// TIA Portal V17 export
// export: Created 2021-12-03T08:08:05.7344229Z, ExportSetting WithDefaults, DisplayName Totally Integrated Automation Portal, DisplayVersion V17, DisplayName TIA Portal Openness, DisplayVersion V17, DisplayName TIA Portal Version Control Interface, DisplayVersion V17, DisplayName STEP 7 Professional, DisplayVersion V17, DisplayName STEP 7 Safety, DisplayVersion V17, DisplayName WinCC Advanced, DisplayVersion V17
VAR_GLOBAL   // PLC tag table "Data_Send"
   CircBrcSts AT %MW100 : Int;   // Автоматические выключатели
   CircBrcSts_0 AT %M100.0 : Bool;
   CircBrcSts_1 AT %M100.1 : Bool;
   CircBrcSts_2 AT %M100.2 : Bool;
   CircBrcSts_3 AT %M100.3 : Bool;
   CircBrcSts_4 AT %M100.4 : Bool;
   CircBrcSts_5 AT %M100.5 : Bool;
   CircBrcSts_6 AT %M100.6 : Bool;
   CircBrcSts_7 AT %M100.7 : Bool;
   CircBrcSts_8 AT %M101.0 : Bool;
   CircBrcSts_9 AT %M101.1 : Bool;
   CircBrcSts_10 AT %M101.2 : Bool;
   CircBrcSts_11 AT %M101.3 : Bool;
   CircBrcSts_12 AT %M101.4 : Bool;
   CircBrcSts_13 AT %M101.5 : Bool;
   CircBrcSts_14 AT %M101.6 : Bool;
   CircBrcSts_15 AT %M101.7 : Bool;
   AccSts AT %MW102 : Int;   // Сигналы с ускорителя
   AccSts_0 AT %M102.0 : Bool;
   AccSts_1 AT %M102.1 : Bool;
   AccSts_2 AT %M102.2 : Bool;
   AccSts_3 AT %M102.3 : Bool;
   AccSts_4 AT %M102.4 : Bool;
   AccSts_5 AT %M102.5 : Bool;
   AccSts_6 AT %M102.6 : Bool;
   AccSts_7 AT %M102.7 : Bool;
   AccSts_8 AT %M103.0 : Bool;
   AccSts_9 AT %M103.1 : Bool;
   AccSts_10 AT %M103.2 : Bool;
   AccSts_11 AT %M103.3 : Bool;
   AccSts_12 AT %M103.4 : Bool;
   AccSts_13 AT %M103.5 : Bool;
   AccSts_14 AT %M103.6 : Bool;
   AccSts_15 AT %M103.7 : Bool;
   P1EmrStp AT %MW104 : Int;   // Аварийный останов Р1
   P1EmrStp_0 AT %M104.0 : Bool;
   P1EmrStp_1 AT %M104.1 : Bool;
   P1EmrStp_2 AT %M104.2 : Bool;
   P2EmrStp AT %MW106 : Int;   // Аварийный останов Р2
   P2EmrStp_0 AT %M106.0 : Bool;
   P2EmrStp_1 AT %M106.1 : Bool;
   P2EmrStp_2 AT %M106.2 : Bool;
   P3EmrStp AT %MW108 : Int;   // Аварийный останов Р3
   P3EmrStp_0 AT %M108.0 : Bool;
   P3EmrStp_1 AT %M108.1 : Bool;
   P3EmrStp_2 AT %M108.2 : Bool;
   AccEmrStp AT %MW110 : Int;   // Аварийный останов от ускорителя
   AccEmrStp_0 AT %M110.0 : Bool;
   AccEmrStp_1 AT %M110.1 : Bool;
   AccEmrStp_2 AT %M110.2 : Bool;
   DosimEmrStp AT %MW112 : Int;   // Аварийный останов от дозиметра
   DosimEmrStp_0 AT %M112.0 : Bool;
   DosimEmrStp_1 AT %M112.1 : Bool;
   DosimEmrStp_2 AT %M112.2 : Bool;
   Cmd AT %MW114 : Int;   // Состояние системы
   Cmd_0 AT %M114.0 : Bool;
   Cmd_1 AT %M114.1 : Bool;
   Cmd_2 AT %M114.2 : Bool;
   Cmd_3 AT %M114.3 : Bool;
   Cmd_4 AT %M114.4 : Bool;
   Cmd_5 AT %M114.5 : Bool;
   Cmd_6 AT %M114.6 : Bool;
   Cmd_7 AT %M114.7 : Bool;
   Cmd_8 AT %M115.0 : Bool;
   Cmd_9 AT %M115.1 : Bool;
   Cmd_10 AT %M115.2 : Bool;
   Cmd_11 AT %M115.3 : Bool;
   Cmd_12 AT %M115.4 : Bool;
   Cmd_13 AT %M115.5 : Bool;
   Cmd_14 AT %M115.6 : Bool;
   Cmd_15 AT %M115.7 : Bool;
   Sft AT %MW116 : Int;   // Состояние систем безопасности
   Sft_0 AT %M116.0 : Bool;
   Sft_1 AT %M116.1 : Bool;
   Sft_2 AT %M116.2 : Bool;
   Sft_3 AT %M116.3 : Bool;
   Sft_4 AT %M116.4 : Bool;
   Sft_5 AT %M116.5 : Bool;
   Sft_6 AT %M116.6 : Bool;
   Sft_7 AT %M116.7 : Bool;
   Sft_8 AT %M117.0 : Bool;
   Sft_9 AT %M117.1 : Bool;
   Sft_10 AT %M117.2 : Bool;
   Sft_11 AT %M117.3 : Bool;
   Sft_12 AT %M117.4 : Bool;
   Sft_13 AT %M117.5 : Bool;
   Sft_14 AT %M117.6 : Bool;
   Sft_15 AT %M117.7 : Bool;
   GnEmStp AT %MW118 : Int;
   GnEmStp_0 AT %M118.0 : Bool;
   GnEmStp_1 AT %M118.1 : Bool;
   GnEmStp_2 AT %M118.2 : Bool;
   Mod400_RlyOn AT %MW120 : Int;
   Mod400_RlyOn_0 AT %M120.0 : Bool;
   Mod400_RlyOn_1 AT %M120.1 : Bool;
   Mod400_RlyOn_2 AT %M120.2 : Bool;
   Mod400_RlyOn_3 AT %M120.3 : Bool;
   Mod400_RlyOn_4 AT %M120.4 : Bool;
   Mod400_RlyOn_5 AT %M120.5 : Bool;
   Mod400_RlyOn_6 AT %M120.6 : Bool;
   Mod400_RlyOn_7 AT %M120.7 : Bool;
   Mod400_RlyOn_8 AT %M121.0 : Bool;
   Mod400_RlyOn_9 AT %M121.1 : Bool;
   Mod400_RlyOn_10 AT %M121.2 : Bool;
   Mod400_RlyOn_11 AT %M121.3 : Bool;
   Mod400_RlyOn_12 AT %M121.4 : Bool;
   Mod400_RlyOn_13 AT %M121.5 : Bool;
   Mod400_RlyOn_14 AT %M121.6 : Bool;
   Mod400_RlyOn_15 AT %M121.7 : Bool;
   Mod230_RlyOn AT %MW122 : Int;
   Mod230_RlyOn_0 AT %M122.0 : Bool;
   Mod230_RlyOn_1 AT %M122.1 : Bool;
   Mod230_RlyOn_2 AT %M122.2 : Bool;
   Mod230_RlyOn_3 AT %M122.3 : Bool;
   Mod230_RlyOn_4 AT %M122.4 : Bool;
   Mod230_RlyOn_5 AT %M122.5 : Bool;
   Mod230_RlyOn_6 AT %M122.6 : Bool;
   Mod230_RlyOn_7 AT %M122.7 : Bool;
   Mod230_RlyOn_8 AT %M123.0 : Bool;
   Mod230_RlyOn_9 AT %M123.1 : Bool;
   Mod230_RlyOn_10 AT %M123.2 : Bool;
   Mod230_RlyOn_11 AT %M123.3 : Bool;
   Mod230_RlyOn_12 AT %M123.4 : Bool;
   Mod230_RlyOn_13 AT %M123.5 : Bool;
   Mod230_RlyOn_14 AT %M123.6 : Bool;
   Mod230_RlyOn_15 AT %M123.7 : Bool;
   Chill_RlyOn AT %MW124 : Int;
   Chill_RlyOn_0 AT %M124.0 : Bool;
   Chill_RlyOn_1 AT %M124.1 : Bool;
   Chill_RlyOn_2 AT %M124.2 : Bool;
   Chill_RlyOn_3 AT %M124.3 : Bool;
   Chill_RlyOn_4 AT %M124.4 : Bool;
   Chill_RlyOn_5 AT %M124.5 : Bool;
   Chill_RlyOn_6 AT %M124.6 : Bool;
   Chill_RlyOn_7 AT %M124.7 : Bool;
   Chill_RlyOn_8 AT %M125.0 : Bool;
   Chill_RlyOn_9 AT %M125.1 : Bool;
   Chill_RlyOn_10 AT %M125.2 : Bool;
   Chill_RlyOn_11 AT %M125.3 : Bool;
   Chill_RlyOn_12 AT %M125.4 : Bool;
   Chill_RlyOn_13 AT %M125.5 : Bool;
   Chill_RlyOn_14 AT %M125.6 : Bool;
   Chill_RlyOn_15 AT %M125.7 : Bool;
   Acc_RlyOn AT %MW126 : Int;
   Acc_RlyOn_0 AT %M126.0 : Bool;
   Acc_RlyOn_1 AT %M126.1 : Bool;
   Acc_RlyOn_2 AT %M126.2 : Bool;
   Acc_RlyOn_3 AT %M126.3 : Bool;
   Acc_RlyOn_4 AT %M126.4 : Bool;
   Acc_RlyOn_5 AT %M126.5 : Bool;
   Acc_RlyOn_6 AT %M126.6 : Bool;
   Acc_RlyOn_7 AT %M126.7 : Bool;
   Acc_RlyOn_8 AT %M127.0 : Bool;
   Acc_RlyOn_9 AT %M127.1 : Bool;
   Acc_RlyOn_10 AT %M127.2 : Bool;
   Acc_RlyOn_11 AT %M127.3 : Bool;
   Acc_RlyOn_12 AT %M127.4 : Bool;
   Acc_RlyOn_13 AT %M127.5 : Bool;
   Acc_RlyOn_14 AT %M127.6 : Bool;
   Acc_RlyOn_15 AT %M127.7 : Bool;
   Conv_RlyOn AT %MW128 : Int;
   Conv_RlyOn_0 AT %M128.0 : Bool;
   Conv_RlyOn_1 AT %M128.1 : Bool;
   Conv_RlyOn_2 AT %M128.2 : Bool;
   Conv_RlyOn_3 AT %M128.3 : Bool;
   Conv_RlyOn_4 AT %M128.4 : Bool;
   Conv_RlyOn_5 AT %M128.5 : Bool;
   Conv_RlyOn_6 AT %M128.6 : Bool;
   Conv_RlyOn_7 AT %M128.7 : Bool;
   Conv_RlyOn_8 AT %M129.0 : Bool;
   Conv_RlyOn_9 AT %M129.1 : Bool;
   Conv_RlyOn_10 AT %M129.2 : Bool;
   Conv_RlyOn_11 AT %M129.3 : Bool;
   Conv_RlyOn_12 AT %M129.4 : Bool;
   Conv_RlyOn_13 AT %M129.5 : Bool;
   Conv_RlyOn_14 AT %M129.6 : Bool;
   Conv_RlyOn_15 AT %M129.7 : Bool;
   ConvSns AT %MW132 : Int;
   ConvSns_0 AT %M132.0 : Bool;
   ConvSns_1 AT %M132.1 : Bool;
   ConvSns_2 AT %M132.2 : Bool;
   ConvSns_3 AT %M132.3 : Bool;
   ConvSns_4 AT %M132.4 : Bool;
   ConvSns_5 AT %M132.5 : Bool;
   ConvSns_6 AT %M132.6 : Bool;
   ConvSns_7 AT %M132.7 : Bool;
   ConvSns_8 AT %M133.0 : Bool;
   ConvSns_9 AT %M133.1 : Bool;
   ConvSns_10 AT %M133.2 : Bool;
   ConvSns_11 AT %M133.3 : Bool;
   ConvSns_12 AT %M133.4 : Bool;
   ConvSns_13 AT %M133.5 : Bool;
   ConvSns_14 AT %M133.6 : Bool;
   ConvSns_15 AT %M133.7 : Bool;
   ScanSeq_Sts AT %MW134 : Int;
   ScanSeq_Sts_0 AT %M134.0 : Bool;
   ScanSeq_Sts_1 AT %M134.1 : Bool;
   ScanSeq_Sts_2 AT %M134.2 : Bool;
   ScanSeq_Sts_3 AT %M134.3 : Bool;
   ScanSeq_Sts_4 AT %M134.4 : Bool;
   ScanSeq_Sts_5 AT %M134.5 : Bool;
   ScanSeq_Sts_6 AT %M134.6 : Bool;
   ScanSeq_Sts_7 AT %M134.7 : Bool;
   ScanSeq_Sts_8 AT %M135.0 : Bool;
   ScanSeq_Sts_9 AT %M135.1 : Bool;
   ScanSeq_Sts_10 AT %M135.2 : Bool;
   ScanSeq_Sts_11 AT %M135.3 : Bool;
   ScanSeq_Sts_12 AT %M135.4 : Bool;
   ScanSeq_Sts_13 AT %M135.5 : Bool;
   ScanSeq_Sts_14 AT %M135.6 : Bool;
   ScanSeq_Sts_15 AT %M135.7 : Bool;
   DetLine_Sts AT %MW136 : Int;
   DetLine_Sts_0 AT %M136.0 : Bool;
   DetLine_Sts_1 AT %M136.1 : Bool;
   DetLine_Sts_2 AT %M136.2 : Bool;
   DetLine_Sts_3 AT %M136.3 : Bool;
   DetLine_Sts_4 AT %M136.4 : Bool;
   DetLine_Sts_5 AT %M136.5 : Bool;
   DetLine_Sts_6 AT %M136.6 : Bool;
   DetLine_Sts_7 AT %M136.7 : Bool;
   DetLine_Sts_8 AT %M137.0 : Bool;
   DetLine_Sts_9 AT %M137.1 : Bool;
   DetLine_Sts_10 AT %M137.2 : Bool;
   DetLine_Sts_11 AT %M137.3 : Bool;
   DetLine_Sts_12 AT %M137.4 : Bool;
   DetLine_Sts_13 AT %M137.5 : Bool;
   DetLine_Sts_14 AT %M137.6 : Bool;
   DetLine_Sts_15 AT %M137.7 : Bool;
   Pwr_All AT %MW138 : Int;
   Pwr_All_0 AT %M138.0 : Bool;
   Pwr_All_1 AT %M138.1 : Bool;
   Pwr_All_2 AT %M138.2 : Bool;
   Pwr_All_3 AT %M138.3 : Bool;
   Pwr_All_4 AT %M138.4 : Bool;
   Pwr_All_5 AT %M138.5 : Bool;
   Pwr_All_6 AT %M138.6 : Bool;
   Pwr_All_7 AT %M138.7 : Bool;
   Pwr_All_8 AT %M139.0 : Bool;
   Pwr_All_9 AT %M139.1 : Bool;
   Pwr_All_10 AT %M139.2 : Bool;
   Pwr_All_11 AT %M139.3 : Bool;
   Pwr_All_12 AT %M139.4 : Bool;
   Pwr_All_13 AT %M139.5 : Bool;
   Pwr_All_14 AT %M139.6 : Bool;
   Pwr_All_15 AT %M139.7 : Bool;
END_VAR
